# EPICS autosave request: i404App/Db/modules_I404.req
#FILE... modules_I404.req

file "I404.req", DEVICE=lsx16a{i404:1}
#file "I404.req", DEVICE=lsx16a{i404:2}
